FUNCTION_BLOCK FB_Beckhoff_EV
VAR_INPUT
END_VAR
VAR_OUTPUT
END_VAR
VAR
END_VAR

END_FUNCTION_BLOCK

(* stored: Version 1.1.0.1, ProductVersion 3.1.4022.18
   POU FB_Beckhoff_EV: Id {69dbe703-9850-4bab-81b1-cfc01666d710}, SpecialFunc None
   Folder Methods: Id {af25a40f-1b5d-4bc9-8db3-3f78b5c85bc1}
   Folder Properties: Id {6d8ca68e-0701-4328-a268-f2b5024f45d0}
   Folder Run: Id {7e75d962-8844-47ae-8e12-11d1abe14ec8} *)
